// TIA Portal V16 export
// export: Created 2023-10-30T22:43:52.8265237Z, ExportSetting WithDefaults, DisplayName Totally Integrated Automation Portal, DisplayVersion V16, DisplayName TIA Portal Version Control Interface, DisplayVersion V16, DisplayName TIA Portal Openness, DisplayVersion V16, DisplayName SINAMICS Startdrive Advanced, DisplayVersion V16, DisplayName SINAMICS Startdrive G130, G150, S120, S150, SINAMICS MV, S210, DisplayVersion V16, DisplayName SINAMICS Startdrive G110M, G120, G120C, G120D, G120P, DisplayVersion V16, DisplayName STEP 7 Professional, DisplayVersion V16, DisplayName STEP 7 Safety, DisplayVersion V16, DisplayName WinCC Professional, DisplayVersion V16
DATA_BLOCK "DB 333"   // DB333
{ S7_Optimized_Access := 'FALSE' }
AUTHOR : AWP_S7P
FAMILY : WEB
VERSION : 1.0
// stored: AutoNumber false, DBAccessibleFromOPCUA true, IsOnlyStoredInLoadMemory false, IsWriteProtectedInAS false
   VAR
      magic { ExternalAccessible := 'False'; ExternalVisible := 'False'; ExternalWritable := 'False'} : DWord := DW#16#41575043;
      consistency_tag { ExternalAccessible := 'False'; ExternalVisible := 'False'; ExternalWritable := 'False'} : DWord := DW#16#24B8E9AC;
      db_version { ExternalAccessible := 'False'; ExternalVisible := 'False'; ExternalWritable := 'False'} : Word := W#16#0001;
      length { ExternalAccessible := 'False'; ExternalVisible := 'False'; ExternalWritable := 'False'} : UInt := 4326;
      pagetab_of { ExternalAccessible := 'False'; ExternalVisible := 'False'; ExternalWritable := 'False'} : UInt := 92;
      pagetab_count { ExternalAccessible := 'False'; ExternalVisible := 'False'; ExternalWritable := 'False'} : UInt := 36;
      excludetab_of { ExternalAccessible := 'False'; ExternalVisible := 'False'; ExternalWritable := 'False'} : UInt := 452;
      excludetab_count { ExternalAccessible := 'False'; ExternalVisible := 'False'; ExternalWritable := 'False'} : UInt := 4;
      fragmentlist_of { ExternalAccessible := 'False'; ExternalVisible := 'False'; ExternalWritable := 'False'} : UInt := 460;
      fragmentlist_count { ExternalAccessible := 'False'; ExternalVisible := 'False'; ExternalWritable := 'False'} : UInt := 55;
      fragmenttab_of { ExternalAccessible := 'False'; ExternalVisible := 'False'; ExternalWritable := 'False'} : UInt := 576;
      fragmenttab_count { ExternalAccessible := 'False'; ExternalVisible := 'False'; ExternalWritable := 'False'} : UInt := 45;
      datatab_of { ExternalAccessible := 'False'; ExternalVisible := 'False'; ExternalWritable := 'False'} : UInt := 1206;
      datatab_count { ExternalAccessible := 'False'; ExternalVisible := 'False'; ExternalWritable := 'False'} : UInt := 30;
      usenametab_of { ExternalAccessible := 'False'; ExternalVisible := 'False'; ExternalWritable := 'False'} : UInt := 1326;
      usenametab_count { ExternalAccessible := 'False'; ExternalVisible := 'False'; ExternalWritable := 'False'} : UInt := 0;
      enumreftab_of { ExternalAccessible := 'False'; ExternalVisible := 'False'; ExternalWritable := 'False'} : UInt := 1326;
      enumreftab_count { ExternalAccessible := 'False'; ExternalVisible := 'False'; ExternalWritable := 'False'} : UInt := 0;
      enumtab_of { ExternalAccessible := 'False'; ExternalVisible := 'False'; ExternalWritable := 'False'} : UInt := 1326;
      enumtab_count { ExternalAccessible := 'False'; ExternalVisible := 'False'; ExternalWritable := 'False'} : UInt := 0;
      textlist_of { ExternalAccessible := 'False'; ExternalVisible := 'False'; ExternalWritable := 'False'} : UInt := 1326;
      textlist_count { ExternalAccessible := 'False'; ExternalVisible := 'False'; ExternalWritable := 'False'} : UInt := 3000;
      language_frag_tab_of { ExternalAccessible := 'False'; ExternalVisible := 'False'; ExternalWritable := 'False'} : UInt := 570;
      language_frag_tab_count { ExternalAccessible := 'False'; ExternalVisible := 'False'; ExternalWritable := 'False'} : UInt := 6;
      application_name { ExternalAccessible := 'False'; ExternalVisible := 'False'; ExternalWritable := 'False'} : UInt := 1;
      application_url { ExternalAccessible := 'False'; ExternalVisible := 'False'; ExternalWritable := 'False'} : UInt := 17;
      application_desc { ExternalAccessible := 'False'; ExternalVisible := 'False'; ExternalWritable := 'False'} : UInt := 34;
      enum_defs_fragment_start { ExternalAccessible := 'False'; ExternalVisible := 'False'; ExternalWritable := 'False'} : UInt := 0;
      enum_defs_fragment_count { ExternalAccessible := 'False'; ExternalVisible := 'False'; ExternalWritable := 'False'} : UInt := 0;
      commandstate { ExternalAccessible := 'False'; ExternalVisible := 'False'; ExternalWritable := 'False'} : Struct
         last_error { ExternalAccessible := 'False'; ExternalVisible := 'False'; ExternalWritable := 'False'} : Int := 0;
         debug_mode { ExternalAccessible := 'False'; ExternalVisible := 'False'; ExternalWritable := 'False'} : Int := 0;
         init { ExternalAccessible := 'False'; ExternalVisible := 'False'; ExternalWritable := 'False'} : Bool := True;
         deactivate { ExternalAccessible := 'False'; ExternalVisible := 'False'; ExternalWritable := 'False'} : Bool := False;
         initializing { ExternalAccessible := 'False'; ExternalVisible := 'False'; ExternalWritable := 'False'} : Bool := False;
         error { ExternalAccessible := 'False'; ExternalVisible := 'False'; ExternalWritable := 'False'} : Bool := False;
         deactivating { ExternalAccessible := 'False'; ExternalVisible := 'False'; ExternalWritable := 'False'} : Bool := False;
         deactivated { ExternalAccessible := 'False'; ExternalVisible := 'False'; ExternalWritable := 'False'} : Bool := False;
         initialized { ExternalAccessible := 'False'; ExternalVisible := 'False'; ExternalWritable := 'False'} : Bool := False;
         reserved1 { ExternalAccessible := 'False'; ExternalVisible := 'False'; ExternalWritable := 'False'} : Bool := False;
         reserved2 { ExternalAccessible := 'False'; ExternalVisible := 'False'; ExternalWritable := 'False'} : Byte := B#16#00;
      END_STRUCT;
      requesttab { ExternalAccessible := 'False'; ExternalVisible := 'False'; ExternalWritable := 'False'} : Array[1..4] of Struct
         page_index { ExternalAccessible := 'False'; ExternalVisible := 'False'; ExternalWritable := 'False'} : UInt;
         fragment_index { ExternalAccessible := 'False'; ExternalVisible := 'False'; ExternalWritable := 'False'} : UInt;
         continue { ExternalAccessible := 'False'; ExternalVisible := 'False'; ExternalWritable := 'False'} : Bool;
         "repeat" { ExternalAccessible := 'False'; ExternalVisible := 'False'; ExternalWritable := 'False'} : Bool;
         abort { ExternalAccessible := 'False'; ExternalVisible := 'False'; ExternalWritable := 'False'} : Bool;
         finish { ExternalAccessible := 'False'; ExternalVisible := 'False'; ExternalWritable := 'False'} : Bool;
         idle { ExternalAccessible := 'False'; ExternalVisible := 'False'; ExternalWritable := 'False'} : Bool;
         waiting { ExternalAccessible := 'False'; ExternalVisible := 'False'; ExternalWritable := 'False'} : Bool;
         sending { ExternalAccessible := 'False'; ExternalVisible := 'False'; ExternalWritable := 'False'} : Bool;
         aborting { ExternalAccessible := 'False'; ExternalVisible := 'False'; ExternalWritable := 'False'} : Bool;
         reserved3 { ExternalAccessible := 'False'; ExternalVisible := 'False'; ExternalWritable := 'False'} : Byte;
      END_STRUCT;
      pagetab { ExternalAccessible := 'False'; ExternalVisible := 'False'; ExternalWritable := 'False'} : Array[1..36] of Struct
         index { ExternalAccessible := 'False'; ExternalVisible := 'False'; ExternalWritable := 'False'} : UInt;
         url { ExternalAccessible := 'False'; ExternalVisible := 'False'; ExternalWritable := 'False'} : UInt;
         mime_type { ExternalAccessible := 'False'; ExternalVisible := 'False'; ExternalWritable := 'False'} : UInt;
         fragment_start { ExternalAccessible := 'False'; ExternalVisible := 'False'; ExternalWritable := 'False'} : UInt;
         fragment_num { ExternalAccessible := 'False'; ExternalVisible := 'False'; ExternalWritable := 'False'} : UInt;
      END_STRUCT;
      excludetab { ExternalAccessible := 'False'; ExternalVisible := 'False'; ExternalWritable := 'False'} : Array[1..4] of UInt;
      fragmentlist { ExternalAccessible := 'False'; ExternalVisible := 'False'; ExternalWritable := 'False'} : Array[1..55] of UInt;
      language_frag_tab { ExternalAccessible := 'False'; ExternalVisible := 'False'; ExternalWritable := 'False'} : Struct
         max_language { ExternalAccessible := 'False'; ExternalVisible := 'False'; ExternalWritable := 'False'} : UInt := 0;
         fragment_count { ExternalAccessible := 'False'; ExternalVisible := 'False'; ExternalWritable := 'False'} : UInt := 0;
         nolang_offset { ExternalAccessible := 'False'; ExternalVisible := 'False'; ExternalWritable := 'False'} : UInt := 0;
      END_STRUCT;
      fragmenttab { ExternalAccessible := 'False'; ExternalVisible := 'False'; ExternalWritable := 'False'} : Array[1..45] of Struct
         fragment_name { ExternalAccessible := 'False'; ExternalVisible := 'False'; ExternalWritable := 'False'} : UInt;
         fragment_type { ExternalAccessible := 'False'; ExternalVisible := 'False'; ExternalWritable := 'False'} : Byte;
         fragment_version { ExternalAccessible := 'False'; ExternalVisible := 'False'; ExternalWritable := 'False'} : Byte;
         content_db { ExternalAccessible := 'False'; ExternalVisible := 'False'; ExternalWritable := 'False'} : UInt;
         content_of { ExternalAccessible := 'False'; ExternalVisible := 'False'; ExternalWritable := 'False'} : UInt;
         content_length { ExternalAccessible := 'False'; ExternalVisible := 'False'; ExternalWritable := 'False'} : UInt;
         data_start { ExternalAccessible := 'False'; ExternalVisible := 'False'; ExternalWritable := 'False'} : UInt;
         data_num { ExternalAccessible := 'False'; ExternalVisible := 'False'; ExternalWritable := 'False'} : UInt;
      END_STRUCT;
      datatab { ExternalAccessible := 'False'; ExternalVisible := 'False'; ExternalWritable := 'False'} : Array[1..30] of Struct
         variable_name { ExternalAccessible := 'False'; ExternalVisible := 'False'; ExternalWritable := 'False'} : UInt;
         direction { ExternalAccessible := 'False'; ExternalVisible := 'False'; ExternalWritable := 'False'} : Int;
      END_STRUCT;
      textlist { ExternalAccessible := 'False'; ExternalVisible := 'False'; ExternalWritable := 'False'} : Array[1..3000] of Byte := 5365727669646F725175616E74756D0076696577735C6C6F67696E2E68746D6C005365727669646F725175616E74756D00494F4431487973745374617475732E68746D6C00746578742F68746D6C00494F44314D6F64652E68746D6C00746578742F68746D6C00494F44315374617475732E68746D6C00746578742F68746D6C00494F4465685374617475732E68746D6C00746578742F68746D6C00494F48756D4431312E68746D6C00746578742F68746D6C00494F48756D443146696E616C5374617475732E68746D6C00746578742F68746D6C00494F48756D4431496E69745374617475732E68746D6C00746578742F68746D6C00494F48756D44314D69645374617475732E68746D6C00746578742F68746D6C00494F48756D44315374617475732E68746D6C00746578742F68746D6C00494F53746172744465682E68746D6C00746578742F68746D6C00494F53746F704465682E68746D6C00746578742F68746D6C00494F54656D7044312E68746D6C00746578742F68746D6C00494F54656D70443146696E616C5374617475732E68746D6C00746578742F68746D6C00494F54656D704431496E69745374617475732E68746D6C00746578742F68746D6C00494F54656D7044314D69645374617475732E68746D6C00746578742F68746D6C00494F54656D7044315374617475732E68746D6C00746578742F68746D6C006E61764261722E68746D6C00746578742F68746D6C00736964654261722E68746D6C00746578742F68746D6C0076696577732F6373732F636F6E74726F6C2E63737300746578742F6373730076696577732F6373732F6C6F67696E2E63737300746578742F6373730076696577732F6373732F6E61765374796C652E63737300746578742F6373730076696577732F6373732F746F67676C655374796C652E63737300746578742F6373730076696577732F64617368626F6172644465682E68746D6C00746578742F68746D6C0076696577732F64617368626F61726448756D44312E68746D6C00746578742F68746D6C0076696577732F64617368626F61726454656D7044312E68746D6C00746578742F68746D6C0076696577732F64617461436F6E74726F6C2E68746D6C00746578742F68746D6C0076696577732F696D672F6C6F676F2E706E6700696D6167652F706E670076696577732F696E6465782E68746D6C00746578742F68746D6C0076696577732F6A732F64617368626F61726448756D44312E6A73006170706C69636174696F6E2F6A6176617363726970740076696577732F6A732F64617368626F61726454656D7044312E6A73006170706C69636174696F6E2F6A6176617363726970740076696577732F6A732F696E6465782E6A73006170706C69636174696F6E2F6A6176617363726970740076696577732F6A732F6A71756572792D332E332E312E6D696E2E6A73006170706C69636174696F6E2F6A6176617363726970740076696577732F6A732F6C6F67696E2E6A73006170706C69636174696F6E2F6A6176617363726970740076696577732F6A732F6E61765363726970742E6A73006170706C69636174696F6E2F6A6176617363726970740076696577732F6A732F736D6F6F74686965322E6A73006170706C69636174696F6E2F6A6176617363726970740076696577732F6C6F67696E2E68746D6C00746578742F68746D6C0076696577732F6373730076696577732F696D670076696577732F6A730076696577730076696577732F6373732F636F6E74726F6C2E6373730076696577732F6373732F6C6F67696E2E6373730076696577732F6373732F6E61765374796C652E6373730076696577732F6373732F746F67676C655374796C652E6373730076696577732F696D672F6C6F676F2E706E670076696577732F696D672F6C6F676F2E706E675F310076696577732F696D672F6C6F676F2E706E675F320076696577732F696D672F6C6F676F2E706E675F330076696577732F6A732F64617368626F61726448756D44312E6A730076696577732F6A732F64617368626F61726454656D7044312E6A730076696577732F6A732F696E6465782E6A730076696577732F6A732F6A71756572792D332E332E312E6D696E2E6A730076696577732F6A732F6A71756572792D332E332E312E6D696E2E6A735F310076696577732F6A732F6C6F67696E2E6A730076696577732F6A732F6E61765363726970742E6A730076696577732F6A732F736D6F6F74686965322E6A730076696577732F64617368626F6172644465682E68746D6C0076696577732F64617368626F6172644465682E68746D6C5F310076696577732F64617368626F61726448756D44312E68746D6C0076696577732F64617368626F61726448756D44312E68746D6C5F310076696577732F64617368626F61726454656D7044312E68746D6C0076696577732F64617368626F61726454656D7044312E68746D6C5F310076696577732F64617461436F6E74726F6C2E68746D6C0076696577732F64617461436F6E74726F6C2E68746D6C5F310076696577732F696E6465782E68746D6C0076696577732F696E6465782E68746D6C5F310076696577732F6C6F67696E2E68746D6C00494F4431487973745374617475732E68746D6C00494F44314D6F64652E68746D6C00494F44315374617475732E68746D6C00494F4465685374617475732E68746D6C00494F48756D4431312E68746D6C00494F48756D443146696E616C5374617475732E68746D6C00494F48756D4431496E69745374617475732E68746D6C00494F48756D44314D69645374617475732E68746D6C00494F48756D44315374617475732E68746D6C00494F53746172744465682E68746D6C00494F53746F704465682E68746D6C00494F54656D7044312E68746D6C00494F54656D70443146696E616C5374617475732E68746D6C00494F54656D704431496E69745374617475732E68746D6C00494F54656D7044314D69645374617475732E68746D6C00494F54656D7044315374617475732E68746D6C006E617642617200736964654261720022416374697661725F44657368696472617461646F722200225365745F506F696E745F44657368696472617461646F722200225365745F506F696E745F48756D6564616422002244657368696472617461646F72220022496E6963696172220022446574656E65722200224D6F646F735F4F7065726163696F6E222E4D6F646F5F5072657365745F443100225365745F506F696E745F44657368696472617461646F72315F496E696369616C2200225365745F506F696E745F44657368696472617461646F72315F496E7465726D656469612200225365745F506F696E745F44657368696472617461646F72315F46696E616C2200225365745F506F696E745F48756D656461645F44315F496E696369616C2200225365745F506F696E745F48756D656461645F44315F496E7465726D656469612200225365745F506F696E745F48756D656461645F44315F46696E616C2200225469656D706F5F486973746572657369735F44312200225469656D706F5F486973746572657369735F44312200224D6F646F735F4F7065726163696F6E222E4D6F646F5F5072657365745F44310022416374697661725F44657368696472617461646F7222002244657368696472617461646F722200224441544F535F5641524941424C4553222E68756D4D6174746500225365745F506F696E745F48756D656461645F44315F46696E616C2200225365745F506F696E745F48756D656461645F44315F496E696369616C2200225365745F506F696E745F48756D656461645F44315F496E7465726D656469612200225365745F506F696E745F48756D65646164220022496E6963696172220022446574656E65722200224441544F535F5641524941424C4553222E74656D704D6174746500225365745F506F696E745F44657368696472617461646F72315F46696E616C2200225365745F506F696E745F44657368696472617461646F72315F496E696369616C2200225365745F506F696E745F44657368696472617461646F72315F496E7465726D656469612200225365745F506F696E745F44657368696472617461646F72220000;
   END_VAR
BEGIN
   requesttab[1..4].page_index := 0;
   requesttab[1..4].fragment_index := 0;
   requesttab[1..4].continue := False;
   requesttab[1..4]."repeat" := False;
   requesttab[1..4].abort := False;
   requesttab[1..4].finish := False;
   requesttab[1..4].idle := False;
   requesttab[1..4].waiting := False;
   requesttab[1..4].sending := False;
   requesttab[1..4].aborting := False;
   requesttab[1..4].reserved3 := B#16#00;
   pagetab[1].index := 1;
   pagetab[2].index := 2;
   pagetab[3].index := 3;
   pagetab[4].index := 4;
   pagetab[5].index := 5;
   pagetab[6].index := 6;
   pagetab[7].index := 7;
   pagetab[8].index := 8;
   pagetab[9].index := 9;
   pagetab[10].index := 10;
   pagetab[11].index := 11;
   pagetab[12].index := 12;
   pagetab[13].index := 13;
   pagetab[14].index := 14;
   pagetab[15].index := 15;
   pagetab[16].index := 16;
   pagetab[17].index := 17;
   pagetab[18].index := 18;
   pagetab[19].index := 19;
   pagetab[20].index := 20;
   pagetab[21].index := 21;
   pagetab[22].index := 22;
   pagetab[23].index := 23;
   pagetab[24].index := 24;
   pagetab[25].index := 25;
   pagetab[26].index := 26;
   pagetab[27].index := 27;
   pagetab[28].index := 28;
   pagetab[29].index := 29;
   pagetab[30].index := 30;
   pagetab[31].index := 31;
   pagetab[32].index := 32;
   pagetab[33].index := 33;
   pagetab[34].index := 34;
   pagetab[35].index := 35;
   pagetab[36].index := 36;
   pagetab[1].url := 50;
   pagetab[2].url := 80;
   pagetab[3].url := 104;
   pagetab[4].url := 130;
   pagetab[5].url := 157;
   pagetab[6].url := 181;
   pagetab[7].url := 215;
   pagetab[8].url := 248;
   pagetab[9].url := 280;
   pagetab[10].url := 309;
   pagetab[11].url := 335;
   pagetab[12].url := 360;
   pagetab[13].url := 384;
   pagetab[14].url := 419;
   pagetab[15].url := 453;
   pagetab[16].url := 486;
   pagetab[17].url := 516;
   pagetab[18].url := 538;
   pagetab[19].url := 561;
   pagetab[20].url := 592;
   pagetab[21].url := 621;
   pagetab[22].url := 653;
   pagetab[23].url := 688;
   pagetab[24].url := 722;
   pagetab[25].url := 758;
   pagetab[26].url := 795;
   pagetab[27].url := 828;
   pagetab[28].url := 857;
   pagetab[29].url := 884;
   pagetab[30].url := 934;
   pagetab[31].url := 985;
   pagetab[32].url := 1026;
   pagetab[33].url := 1078;
   pagetab[34].url := 1119;
   pagetab[35].url := 1164;
   pagetab[36].url := 1209;
   pagetab[1].mime_type := 70;
   pagetab[2].mime_type := 94;
   pagetab[3].mime_type := 120;
   pagetab[4].mime_type := 147;
   pagetab[5].mime_type := 171;
   pagetab[6].mime_type := 205;
   pagetab[7].mime_type := 238;
   pagetab[8].mime_type := 270;
   pagetab[9].mime_type := 299;
   pagetab[10].mime_type := 325;
   pagetab[11].mime_type := 350;
   pagetab[12].mime_type := 374;
   pagetab[13].mime_type := 409;
   pagetab[14].mime_type := 443;
   pagetab[15].mime_type := 476;
   pagetab[16].mime_type := 506;
   pagetab[17].mime_type := 528;
   pagetab[18].mime_type := 551;
   pagetab[19].mime_type := 583;
   pagetab[20].mime_type := 612;
   pagetab[21].mime_type := 644;
   pagetab[22].mime_type := 679;
   pagetab[23].mime_type := 712;
   pagetab[24].mime_type := 748;
   pagetab[25].mime_type := 785;
   pagetab[26].mime_type := 818;
   pagetab[27].mime_type := 847;
   pagetab[28].mime_type := 874;
   pagetab[29].mime_type := 911;
   pagetab[30].mime_type := 962;
   pagetab[31].mime_type := 1003;
   pagetab[32].mime_type := 1055;
   pagetab[33].mime_type := 1096;
   pagetab[34].mime_type := 1141;
   pagetab[35].mime_type := 1186;
   pagetab[36].mime_type := 1226;
   pagetab[1].fragment_start := 1;
   pagetab[2].fragment_start := 2;
   pagetab[3].fragment_start := 3;
   pagetab[4].fragment_start := 4;
   pagetab[5].fragment_start := 5;
   pagetab[6].fragment_start := 6;
   pagetab[7].fragment_start := 7;
   pagetab[8].fragment_start := 8;
   pagetab[9].fragment_start := 9;
   pagetab[10].fragment_start := 10;
   pagetab[11].fragment_start := 11;
   pagetab[12].fragment_start := 12;
   pagetab[13].fragment_start := 13;
   pagetab[14].fragment_start := 14;
   pagetab[15].fragment_start := 15;
   pagetab[16].fragment_start := 16;
   pagetab[17].fragment_start := 17;
   pagetab[18].fragment_start := 18;
   pagetab[19].fragment_start := 19;
   pagetab[20].fragment_start := 20;
   pagetab[21].fragment_start := 21;
   pagetab[22].fragment_start := 22;
   pagetab[23].fragment_start := 23;
   pagetab[24].fragment_start := 27;
   pagetab[25].fragment_start := 31;
   pagetab[26].fragment_start := 35;
   pagetab[27].fragment_start := 39;
   pagetab[28].fragment_start := 43;
   pagetab[29].fragment_start := 47;
   pagetab[30].fragment_start := 48;
   pagetab[31].fragment_start := 49;
   pagetab[32].fragment_start := 50;
   pagetab[33].fragment_start := 52;
   pagetab[34].fragment_start := 53;
   pagetab[35].fragment_start := 54;
   pagetab[36].fragment_start := 55;
   pagetab[1..22].fragment_num := 1;
   pagetab[23..28].fragment_num := 4;
   pagetab[29..31].fragment_num := 1;
   pagetab[32].fragment_num := 2;
   pagetab[33..36].fragment_num := 1;
   excludetab[1] := 1236;
   excludetab[2] := 1246;
   excludetab[3] := 1256;
   excludetab[4] := 1265;
   fragmentlist[1] := 28;
   fragmentlist[2] := 29;
   fragmentlist[3] := 30;
   fragmentlist[4] := 31;
   fragmentlist[5] := 32;
   fragmentlist[6] := 33;
   fragmentlist[7] := 34;
   fragmentlist[8] := 35;
   fragmentlist[9] := 36;
   fragmentlist[10] := 37;
   fragmentlist[11] := 38;
   fragmentlist[12] := 39;
   fragmentlist[13] := 40;
   fragmentlist[14] := 41;
   fragmentlist[15] := 42;
   fragmentlist[16] := 43;
   fragmentlist[17] := 44;
   fragmentlist[18] := 45;
   fragmentlist[19] := 1;
   fragmentlist[20] := 2;
   fragmentlist[21] := 3;
   fragmentlist[22] := 4;
   fragmentlist[23] := 17;
   fragmentlist[24] := 44;
   fragmentlist[25] := 45;
   fragmentlist[26] := 18;
   fragmentlist[27] := 19;
   fragmentlist[28] := 44;
   fragmentlist[29] := 45;
   fragmentlist[30] := 20;
   fragmentlist[31] := 21;
   fragmentlist[32] := 44;
   fragmentlist[33] := 45;
   fragmentlist[34] := 22;
   fragmentlist[35] := 23;
   fragmentlist[36] := 44;
   fragmentlist[37] := 45;
   fragmentlist[38] := 24;
   fragmentlist[39] := 5;
   fragmentlist[40] := 6;
   fragmentlist[41] := 7;
   fragmentlist[42] := 8;
   fragmentlist[43] := 25;
   fragmentlist[44] := 44;
   fragmentlist[45] := 45;
   fragmentlist[46] := 26;
   fragmentlist[47] := 9;
   fragmentlist[48] := 10;
   fragmentlist[49] := 11;
   fragmentlist[50] := 12;
   fragmentlist[51] := 13;
   fragmentlist[52] := 14;
   fragmentlist[53] := 15;
   fragmentlist[54] := 16;
   fragmentlist[55] := 27;
   fragmenttab[1].fragment_name := 1271;
   fragmenttab[2].fragment_name := 1293;
   fragmenttab[3].fragment_name := 1313;
   fragmenttab[4].fragment_name := 1336;
   fragmenttab[5].fragment_name := 1362;
   fragmenttab[6].fragment_name := 1381;
   fragmenttab[7].fragment_name := 1402;
   fragmenttab[8].fragment_name := 1423;
   fragmenttab[9].fragment_name := 1444;
   fragmenttab[10].fragment_name := 1471;
   fragmenttab[11].fragment_name := 1499;
   fragmenttab[12].fragment_name := 1517;
   fragmenttab[13].fragment_name := 1546;
   fragmenttab[14].fragment_name := 1577;
   fragmenttab[15].fragment_name := 1595;
   fragmenttab[16].fragment_name := 1617;
   fragmenttab[17].fragment_name := 1639;
   fragmenttab[18].fragment_name := 1663;
   fragmenttab[19].fragment_name := 1689;
   fragmenttab[20].fragment_name := 1715;
   fragmenttab[21].fragment_name := 1743;
   fragmenttab[22].fragment_name := 1770;
   fragmenttab[23].fragment_name := 1799;
   fragmenttab[24].fragment_name := 1822;
   fragmenttab[25].fragment_name := 1847;
   fragmenttab[26].fragment_name := 1864;
   fragmenttab[27].fragment_name := 1883;
   fragmenttab[28].fragment_name := 1900;
   fragmenttab[29].fragment_name := 1920;
   fragmenttab[30].fragment_name := 1934;
   fragmenttab[31].fragment_name := 1950;
   fragmenttab[32].fragment_name := 1967;
   fragmenttab[33].fragment_name := 1981;
   fragmenttab[34].fragment_name := 2005;
   fragmenttab[35].fragment_name := 2028;
   fragmenttab[36].fragment_name := 2050;
   fragmenttab[37].fragment_name := 2069;
   fragmenttab[38].fragment_name := 2085;
   fragmenttab[39].fragment_name := 2100;
   fragmenttab[40].fragment_name := 2114;
   fragmenttab[41].fragment_name := 2139;
   fragmenttab[42].fragment_name := 2163;
   fragmenttab[43].fragment_name := 2186;
   fragmenttab[44].fragment_name := 2206;
   fragmenttab[45].fragment_name := 2213;
   fragmenttab[1..45].fragment_type := B#16#00;
   fragmenttab[1..45].fragment_version := B#16#00;
   fragmenttab[1..4].content_db := 334;
   fragmenttab[5].content_db := 335;
   fragmenttab[6].content_db := 336;
   fragmenttab[7].content_db := 337;
   fragmenttab[8..11].content_db := 338;
   fragmenttab[12].content_db := 339;
   fragmenttab[13..15].content_db := 340;
   fragmenttab[16..25].content_db := 341;
   fragmenttab[26..43].content_db := 342;
   fragmenttab[44..45].content_db := 334;
   fragmenttab[1].content_of := 1622;
   fragmenttab[2].content_of := 2684;
   fragmenttab[3].content_of := 3088;
   fragmenttab[4].content_of := 7122;
   fragmenttab[5..8].content_of := 8;
   fragmenttab[9].content_of := 10854;
   fragmenttab[10].content_of := 13240;
   fragmenttab[11].content_of := 14804;
   fragmenttab[12..13].content_of := 8;
   fragmenttab[14].content_of := 21410;
   fragmenttab[15].content_of := 22558;
   fragmenttab[16].content_of := 8;
   fragmenttab[17].content_of := 46036;
   fragmenttab[18].content_of := 48330;
   fragmenttab[19].content_of := 49986;
   fragmenttab[20].content_of := 51444;
   fragmenttab[21].content_of := 52014;
   fragmenttab[22].content_of := 53474;
   fragmenttab[23].content_of := 54046;
   fragmenttab[24].content_of := 58890;
   fragmenttab[25].content_of := 62442;
   fragmenttab[26].content_of := 8;
   fragmenttab[27].content_of := 6822;
   fragmenttab[28].content_of := 10574;
   fragmenttab[29].content_of := 10756;
   fragmenttab[30].content_of := 10942;
   fragmenttab[31].content_of := 11120;
   fragmenttab[32].content_of := 11292;
   fragmenttab[33].content_of := 11472;
   fragmenttab[34].content_of := 11664;
   fragmenttab[35].content_of := 11856;
   fragmenttab[36].content_of := 12050;
   fragmenttab[37].content_of := 12228;
   fragmenttab[38].content_of := 12392;
   fragmenttab[39].content_of := 12556;
   fragmenttab[40].content_of := 12736;
   fragmenttab[41].content_of := 12932;
   fragmenttab[42].content_of := 13130;
   fragmenttab[43].content_of := 13330;
   fragmenttab[44].content_of := 8;
   fragmenttab[45].content_of := 384;
   fragmenttab[1].content_length := 1061;
   fragmenttab[2].content_length := 403;
   fragmenttab[3].content_length := 4034;
   fragmenttab[4].content_length := 1146;
   fragmenttab[5..7].content_length := 65526;
   fragmenttab[8].content_length := 10845;
   fragmenttab[9].content_length := 2386;
   fragmenttab[10].content_length := 1564;
   fragmenttab[11].content_length := 6294;
   fragmenttab[12].content_length := 65526;
   fragmenttab[13].content_length := 21401;
   fragmenttab[14].content_length := 1148;
   fragmenttab[15].content_length := 149;
   fragmenttab[16].content_length := 46027;
   fragmenttab[17].content_length := 2294;
   fragmenttab[18].content_length := 1656;
   fragmenttab[19].content_length := 1457;
   fragmenttab[20].content_length := 570;
   fragmenttab[21].content_length := 1460;
   fragmenttab[22].content_length := 571;
   fragmenttab[23].content_length := 4843;
   fragmenttab[24].content_length := 3552;
   fragmenttab[25].content_length := 1448;
   fragmenttab[26].content_length := 6814;
   fragmenttab[27].content_length := 3752;
   fragmenttab[28].content_length := 181;
   fragmenttab[29].content_length := 185;
   fragmenttab[30].content_length := 178;
   fragmenttab[31].content_length := 171;
   fragmenttab[32].content_length := 179;
   fragmenttab[33].content_length := 191;
   fragmenttab[34].content_length := 192;
   fragmenttab[35].content_length := 194;
   fragmenttab[36].content_length := 177;
   fragmenttab[37].content_length := 164;
   fragmenttab[38].content_length := 163;
   fragmenttab[39].content_length := 180;
   fragmenttab[40].content_length := 196;
   fragmenttab[41].content_length := 197;
   fragmenttab[42].content_length := 199;
   fragmenttab[43].content_length := 184;
   fragmenttab[44].content_length := 375;
   fragmenttab[45].content_length := 1237;
   fragmenttab[1..24].data_start := 0;
   fragmenttab[25].data_start := 1;
   fragmenttab[26..27].data_start := 0;
   fragmenttab[28].data_start := 15;
   fragmenttab[29].data_start := 16;
   fragmenttab[30].data_start := 17;
   fragmenttab[31].data_start := 18;
   fragmenttab[32].data_start := 19;
   fragmenttab[33].data_start := 20;
   fragmenttab[34].data_start := 21;
   fragmenttab[35].data_start := 22;
   fragmenttab[36].data_start := 23;
   fragmenttab[37].data_start := 24;
   fragmenttab[38].data_start := 25;
   fragmenttab[39].data_start := 26;
   fragmenttab[40].data_start := 27;
   fragmenttab[41].data_start := 28;
   fragmenttab[42].data_start := 29;
   fragmenttab[43].data_start := 30;
   fragmenttab[44..45].data_start := 0;
   fragmenttab[1..24].data_num := 0;
   fragmenttab[25].data_num := 14;
   fragmenttab[26..27].data_num := 0;
   fragmenttab[28..43].data_num := 1;
   fragmenttab[44..45].data_num := 0;
   datatab[1].variable_name := 2221;
   datatab[2].variable_name := 2245;
   datatab[3].variable_name := 2271;
   datatab[4].variable_name := 2291;
   datatab[5].variable_name := 2307;
   datatab[6].variable_name := 2317;
   datatab[7].variable_name := 2327;
   datatab[8].variable_name := 2360;
   datatab[9].variable_name := 2395;
   datatab[10].variable_name := 2433;
   datatab[11].variable_name := 2466;
   datatab[12].variable_name := 2497;
   datatab[13].variable_name := 2531;
   datatab[14].variable_name := 2560;
   datatab[15].variable_name := 2583;
   datatab[16].variable_name := 2606;
   datatab[17].variable_name := 2639;
   datatab[18].variable_name := 2663;
   datatab[19].variable_name := 2679;
   datatab[20].variable_name := 2706;
   datatab[21].variable_name := 2735;
   datatab[22].variable_name := 2766;
   datatab[23].variable_name := 2800;
   datatab[24].variable_name := 2820;
   datatab[25].variable_name := 2830;
   datatab[26].variable_name := 2840;
   datatab[27].variable_name := 2868;
   datatab[28].variable_name := 2901;
   datatab[29].variable_name := 2936;
   datatab[30].variable_name := 2974;
   datatab[1..14].direction := 2;
   datatab[15..30].direction := 3;
END_DATA_BLOCK
